Staubli VAL3: CheckRobPos.pgx

program CheckRobPos(joint x_jRef (dimensions=1), bool& x_bStatus (dimensions=1))
  local joint l_j
  local num l_nErr
begin
  //判断当前机器人的位置状态
  //x_jRef:参考位置
  //x_bStatus:
  //--true:机器人在x_jRef
  //--false:机器人不在x_jRef
  l_nErr=0.05
  l_j=herej()
  x_bStatus=false
  if abs(l_j-x_jRef)<{l_nErr,l_nErr,l_nErr,l_nErr,l_nErr,l_nErr}
    x_bStatus=true
  endIf
end
